{region '#Template'}
	{attribute 'Version' := '1.2.0.0'}
	{attribute 'Tags' := '"LCID": "1031", "Text": "DUT, Plant, AC, Setpoint"'}
	{attribute 'Tags' := '"LCID": "1033", "Text": "DUT, Plant, AC, Setpoint"'}
	{attribute 'Description' := '"LCID": "1031", "Text": "Auswahl Sollwert Energie Rückgewinnung"'}
	{attribute 'Description' := '"LCID": "1033", "Text": "Selection setpoint energy recovery"'}
{endregion}

{attribute 'qualified_only'}
TYPE E_BA_AC_SelSpErc :
(
	eAction				:= 1,	//	E_BA_Action.eDirect = SpCol, E_BA_Action.eReverse = SpHtg, 
	eAverageHtgCol		:= 2	
) UDINT;
END_TYPE

(* stored: Version 1.1.0.1, ProductVersion 3.1.4024.9
   DUT E_BA_AC_SelSpErc: Id {c6da13cd-5fd0-4d28-8cfa-3c757560a3dd} *)
